LIN {X 0,Y 227.562,Z 874.921,A -85,B 0,C 180,E1 18435.228,E2 18435.228} C_VEL
LIN {X 0,Y 232.413,Z 908.174,A -85,B 0,C 180,E1 18441.181,E2 18441.181} C_VEL
LIN {X 0,Y 223.238,Z 943.271,A -85,B 0,C 180,E1 18449.512,E2 18449.512} C_VEL
LIN {X 0,Y 216.658,Z 965.158,A -85,B 0,C 180,E1 18460.084,E2 18460.084} C_VEL
LIN {X 0,Y 215.346,Z 974.266,A -85,B 0,C 180,E1 18472.803,E2 18472.803} C_VEL
LIN {X 0,Y 221.79,Z 968.351,A -85,B 0,C 180,E1 18485.562,E2 18485.562} C_VEL
LIN {X 0,Y 234.33,Z 948.382,A -85,B 0,C 180,E1 18496.092,E2 18496.092} C_VEL
LIN {X 0,Y 246.199,Z 920.964,A -85,B 0,C 180,E1 18503.2,E2 18503.2} C_VEL
LIN {X 0,Y 242.131,Z 889.578,A -85,B 0,C 180,E1 18511.964,E2 18511.964} C_VEL
LIN {X 0,Y 229.382,Z 860.327,A -85,B 0,C 180,E1 18522.556,E2 18522.556} C_VEL
LIN {X 0,Y 219.392,Z 845.564,A -85,B 0,C 180,E1 18532.052,E2 18532.052} C_VEL
LIN {X 0,Y 215.629,Z 839.103,A -85,B 0,C 180,E1 18538.996,E2 18538.996} C_VEL
LIN {X 0,Y 216.706,Z 841.817,A -85,B 0,C 180,E1 18553.322,E2 18553.322} C_VEL
LIN {X 0,Y 226.196,Z 855.249,A -85,B 0,C 180,E1 18564.093,E2 18564.093} C_VEL
LIN {X 0,Y 243.066,Z 883.319,A -85,B 0,C 180,E1 18574.736,E2 18574.736} C_VEL
LIN {X 0,Y 255.06,Z 918.124,A -85,B 0,C 180,E1 18582.6,E2 18582.6} C_VEL
LIN {X 0,Y 254.028,Z 931.092,A -85,B 0,C 180,E1 18584.355,E2 18584.355} C_VEL
LIN {X 0,Y 237.373,Z 975.39,A -85,B 0,C 180,E1 18590.854,E2 18590.854} C_VEL
LIN {X 0,Y 221.129,Z 1010.154,A -85,B 0,C 180,E1 18601.29,E2 18601.29} C_VEL
LIN {X 0,Y 213.42,Z 1031.37,A -85,B 0,C 180,E1 18614.546,E2 18614.546} C_VEL
LIN {X 0,Y 214.183,Z 1038.324,A -85,B 0,C 180,E1 18627.971,E2 18627.971} C_VEL
LIN {X 0,Y 213.62,Z 1033.071,A -85,B 0,C 180,E1 18638.747,E2 18638.747} C_VEL
LIN {X 0,Y 215.705,Z 1013.058,A -85,B 0,C 180,E1 18651.676,E2 18651.676} C_VEL
LIN {X 0,Y 225.346,Z 978.895,A -85,B 0,C 180,E1 18662.658,E2 18662.658} C_VEL
LIN {X 0,Y 237.301,Z 933.937,A -85,B 0,C 180,E1 18670.068,E2 18670.068} C_VEL
LIN {X 0,Y 239.733,Z 912.196,A -85,B 0,C 180,E1 18672.372,E2 18672.372} C_VEL
LIN {X 0,Y 223.495,Z 863.245,A -85,B 0,C 180,E1 18678.375,E2 18678.375} C_VEL
LIN {X 0,Y 208.076,Z 831.81,A -85,B 0,C 180,E1 18683.175,E2 18683.175} C_VEL
LIN {X 0,Y 208.641,Z 831.81,A -85,B 0,C 180,E1 18696.413,E2 18696.413} C_VEL
LIN {X 0,Y 209.995,Z 831.81,A -85,B 0,C 180,E1 18709.587,E2 18709.587} C_VEL
LIN {X 0,Y 211.06,Z 831.81,A -85,B 0,C 180,E1 18722.056,E2 18722.056} C_VEL
LIN {X 0,Y 209.619,Z 831.81,A -85,B 0,C 180,E1 18734.674,E2 18734.674} C_VEL
LIN {X 0,Y 208.453,Z 831.81,A -85,B 0,C 180,E1 18748.239,E2 18748.239} C_VEL
LIN {X 0,Y 207.773,Z 831.81,A -85,B 0,C 180,E1 18755.093,E2 18755.093} C_VEL
LIN {X 0,Y 199.619,Z 831.81,A -85,B 0,C 180,E1 18764.876,E2 18764.876} C_VEL
LIN {X 0,Y 200.129,Z 831.81,A -85,B 0,C 180,E1 18780.692,E2 18780.692} C_VEL
LIN {X 0,Y 200.595,Z 833.153,A -85,B 0,C 180,E1 18786.258,E2 18786.258} C_VEL
LIN {X 0,Y 220.002,Z 874.825,A -85,B 0,C 180,E1 18793.82,E2 18793.82} C_VEL
LIN {X 0,Y 225.22,Z 909.27,A -85,B 0,C 180,E1 18800.302,E2 18800.302} C_VEL
LIN {X 0,Y 215.598,Z 944.601,A -85,B 0,C 180,E1 18808.991,E2 18808.991} C_VEL
LIN {X 0,Y 208.485,Z 967.346,A -85,B 0,C 180,E1 18820.692,E2 18820.692} C_VEL
LIN {X 0,Y 207.716,Z 975.562,A -85,B 0,C 180,E1 18834.047,E2 18834.047} C_VEL
LIN {X 0,Y 214.927,Z 969.025,A -85,B 0,C 180,E1 18846.881,E2 18846.881} C_VEL
LIN {X 0,Y 228.472,Z 948.449,A -85,B 0,C 180,E1 18857.625,E2 18857.625} C_VEL
LIN {X 0,Y 239.818,Z 923.429,A -85,B 0,C 180,E1 18864.258,E2 18864.258} C_VEL
LIN {X 0,Y 236.55,Z 893.1,A -85,B 0,C 180,E1 18873.318,E2 18873.318} C_VEL
LIN {X 0,Y 225.614,Z 866.279,A -85,B 0,C 180,E1 18883.894,E2 18883.894} C_VEL
LIN {X 0,Y 217.441,Z 852.723,A -85,B 0,C 180,E1 18893.114,E2 18893.114} C_VEL
LIN {X 0,Y 214.592,Z 847.026,A -85,B 0,C 180,E1 18898.991,E2 18898.991} C_VEL
LIN {X 0,Y 215.401,Z 849.582,A -85,B 0,C 180,E1 18912.822,E2 18912.822} C_VEL
LIN {X 0,Y 224.366,Z 863.156,A -85,B 0,C 180,E1 18923.623,E2 18923.623} C_VEL
LIN {X 0,Y 239.322,Z 890.023,A -85,B 0,C 180,E1 18934.117,E2 18934.117} C_VEL
LIN {X 0,Y 249.469,Z 923.65,A -85,B 0,C 180,E1 18942.061,E2 18942.061} C_VEL
LIN {X 0,Y 234.402,Z 967.505,A -85,B 0,C 180,E1 18948.127,E2 18948.127} C_VEL
LIN {X 0,Y 217.225,Z 1002.987,A -85,B 0,C 180,E1 18957.642,E2 18957.642} C_VEL
LIN {X 0,Y 206.636,Z 1026.774,A -85,B 0,C 180,E1 18970.703,E2 18970.703} C_VEL
LIN {X 0,Y 205.698,Z 1036.793,A -85,B 0,C 180,E1 18984.937,E2 18984.937} C_VEL
LIN {X 0,Y 205.898,Z 1033.928,A -85,B 0,C 180,E1 18996.348,E2 18996.348} C_VEL
LIN {X 0,Y 206.967,Z 1016.698,A -85,B 0,C 180,E1 19009.824,E2 19009.824} C_VEL
LIN {X 0,Y 215.978,Z 984.595,A -85,B 0,C 180,E1 19021.802,E2 19021.802} C_VEL
LIN {X 0,Y 228.47,Z 941.098,A -85,B 0,C 180,E1 19030.075,E2 19030.075} C_VEL
LIN {X 0,Y 232.456,Z 913.301,A -85,B 0,C 180,E1 19033.274,E2 19033.274} C_VEL
LIN {X 0,Y 216.734,Z 865.176,A -85,B 0,C 180,E1 19039.626,E2 19039.626} C_VEL
LIN {X 0,Y 200.024,Z 831.81,A -85,B 0,C 180,E1 19045.311,E2 19045.311} C_VEL
LIN {X 0,Y 201.036,Z 831.81,A -85,B 0,C 180,E1 19060.663,E2 19060.663} C_VEL
LIN {X 0,Y 202.402,Z 831.81,A -85,B 0,C 180,E1 19073.538,E2 19073.538} C_VEL
LIN {X 0,Y 202.406,Z 831.81,A -85,B 0,C 180,E1 19086.453,E2 19086.453} C_VEL
LIN {X 0,Y 201.019,Z 831.81,A -85,B 0,C 180,E1 19099.856,E2 19099.856} C_VEL
LIN {X 0,Y 199.779,Z 831.81,A -85,B 0,C 180,E1 19115.035,E2 19115.035} C_VEL
LIN {X 0,Y 199.619,Z 831.81,A -85,B 0,C 180,E1 19124.876,E2 19124.876} C_VEL
LIN {X 0,Y 191.641,Z 831.81,A -85,B 0,C 180,E1 19135.041,E2 19135.041} C_VEL
LIN {X 0,Y 192.321,Z 833.227,A -85,B 0,C 180,E1 19144.01,E2 19144.01} C_VEL
LIN {X 0,Y 212.038,Z 873.85,A -85,B 0,C 180,E1 19152.114,E2 19152.114} C_VEL
LIN {X 0,Y 218.056,Z 907.218,A -85,B 0,C 180,E1 19158.702,E2 19158.702} C_VEL
LIN {X 0,Y 210.506,Z 938.161,A -85,B 0,C 180,E1 19165.865,E2 19165.865} C_VEL
LIN {X 0,Y 202.25,Z 962.969,A -85,B 0,C 180,E1 19176.462,E2 19176.462} C_VEL
LIN {X 0,Y 199.165,Z 975.841,A -85,B 0,C 180,E1 19190.051,E2 19190.051} C_VEL
LIN {X 0,Y 204.368,Z 973.813,A -85,B 0,C 180,E1 19203.842,E2 19203.842} C_VEL
LIN {X 0,Y 217.789,Z 956.53,A -85,B 0,C 180,E1 19216.152,E2 19216.152} C_VEL
LIN {X 0,Y 233.487,Z 926.207,A -85,B 0,C 180,E1 19225.271,E2 19225.271} C_VEL
LIN {X 0,Y 231.391,Z 897.943,A -85,B 0,C 180,E1 19234.249,E2 19234.249} C_VEL
LIN {X 0,Y 222.035,Z 872.175,A -85,B 0,C 180,E1 19245.152,E2 19245.152} C_VEL
LIN {X 0,Y 215.105,Z 859.024,A -85,B 0,C 180,E1 19254.818,E2 19254.818} C_VEL
LIN {X 0,Y 213.156,Z 854.83,A -85,B 0,C 180,E1 19260.004,E2 19260.004} C_VEL
LIN {X 0,Y 214.206,Z 857.664,A -85,B 0,C 180,E1 19272.602,E2 19272.602} C_VEL
LIN {X 0,Y 222.658,Z 871.543,A -85,B 0,C 180,E1 19283.498,E2 19283.498} C_VEL
LIN {X 0,Y 235.877,Z 897.817,A -85,B 0,C 180,E1 19293.883,E2 19293.883} C_VEL
LIN {X 0,Y 243.66,Z 928.776,A -85,B 0,C 180,E1 19301.455,E2 19301.455} C_VEL
LIN {X 0,Y 225.466,Z 973.136,A -85,B 0,C 180,E1 19308.014,E2 19308.014} C_VEL
LIN {X 0,Y 207.536,Z 1007.322,A -85,B 0,C 180,E1 19318.602,E2 19318.602} C_VEL
LIN {X 0,Y 198.142,Z 1027.993,A -85,B 0,C 180,E1 19332.014,E2 19332.014} C_VEL
LIN {X 0,Y 197.604,Z 1035.315,A -85,B 0,C 180,E1 19343.386,E2 19343.386} C_VEL
LIN {X 0,Y 198.026,Z 1033.573,A -85,B 0,C 180,E1 19354.984,E2 19354.984} C_VEL
LIN {X 0,Y 198.809,Z 1017.493,A -85,B 0,C 180,E1 19369.18,E2 19369.18} C_VEL
LIN {X 0,Y 207.283,Z 987.806,A -85,B 0,C 180,E1 19381.442,E2 19381.442} C_VEL
LIN {X 0,Y 219.997,Z 945.926,A -85,B 0,C 180,E1 19390.293,E2 19390.293} C_VEL
LIN {X 0,Y 225.514,Z 915.954,A -85,B 0,C 180,E1 19394.003,E2 19394.003} C_VEL
LIN {X 0,Y 210.731,Z 868.772,A -85,B 0,C 180,E1 19400.705,E2 19400.705} C_VEL
LIN {X 0,Y 191.908,Z 831.81,A -85,B 0,C 180,E1 19407.681,E2 19407.681} C_VEL
LIN {X 0,Y 193.242,Z 831.81,A -85,B 0,C 180,E1 19424.041,E2 19424.041} C_VEL
LIN {X 0,Y 194.824,Z 831.81,A -85,B 0,C 180,E1 19437.763,E2 19437.763} C_VEL
LIN {X 0,Y 193.764,Z 831.81,A -85,B 0,C 180,E1 19451.763,E2 19451.763} C_VEL
LIN {X 0,Y 192.436,Z 831.81,A -85,B 0,C 180,E1 19465.701,E2 19465.701} C_VEL
LIN {X 0,Y 191.599,Z 831.81,A -85,B 0,C 180,E1 19482.314,E2 19482.314} C_VEL
LIN {X 0,Y 191.641,Z 831.81,A -85,B 0,C 180,E1 19495.041,E2 19495.041} C_VEL
LIN {X 0,Y 183.76,Z 831.81,A -85,B 0,C 180,E1 19499.036,E2 19499.036} C_VEL
LIN {X 0,Y 184.366,Z 834.043,A -85,B 0,C 180,E1 19501.623,E2 19501.623} C_VEL
LIN {X 0,Y 204.05,Z 872.307,A -85,B 0,C 180,E1 19510.187,E2 19510.187} C_VEL
LIN {X 0,Y 211.019,Z 906.88,A -85,B 0,C 180,E1 19517.363,E2 19517.363} C_VEL
LIN {X 0,Y 204.912,Z 934.231,A -85,B 0,C 180,E1 19523.621,E2 19523.621} C_VEL
LIN {X 0,Y 195.354,Z 961.456,A -85,B 0,C 180,E1 19534.455,E2 19534.455} C_VEL
LIN {X 0,Y 191.182,Z 976.246,A -85,B 0,C 180,E1 19548.467,E2 19548.467} C_VEL
LIN {X 0,Y 195.705,Z 976.136,A -85,B 0,C 180,E1 19562.873,E2 19562.873} C_VEL
LIN {X 0,Y 208.443,Z 961.663,A -85,B 0,C 180,E1 19575.466,E2 19575.466} C_VEL
LIN {X 0,Y 225.666,Z 934.091,A -85,B 0,C 180,E1 19584.848,E2 19584.848} C_VEL
LIN {X 0,Y 227.198,Z 909.123,A -85,B 0,C 180,E1 19592.935,E2 19592.935} C_VEL
LIN {X 0,Y 220.603,Z 883.227,A -85,B 0,C 180,E1 19603.518,E2 19603.518} C_VEL
LIN {X 0,Y 213.521,Z 867.423,A -85,B 0,C 180,E1 19614.523,E2 19614.523} C_VEL
LIN {X 0,Y 211.564,Z 862.576,A -85,B 0,C 180,E1 19621.051,E2 19621.051} C_VEL
LIN {X 0,Y 212.721,Z 865.53,A -85,B 0,C 180,E1 19632.238,E2 19632.238} C_VEL
LIN {X 0,Y 220.513,Z 879.568,A -85,B 0,C 180,E1 19643.316,E2 19643.316} C_VEL
LIN {X 0,Y 232.182,Z 905.731,A -85,B 0,C 180,E1 19653.756,E2 19653.756} C_VEL
LIN {X 0,Y 236.869,Z 933.02,A -85,B 0,C 180,E1 19660.477,E2 19660.477} C_VEL
LIN {X 0,Y 217.79,Z 975.94,A -85,B 0,C 180,E1 19667.34,E2 19667.34} C_VEL
LIN {X 0,Y 199.319,Z 1008.691,A -85,B 0,C 180,E1 19678.438,E2 19678.438} C_VEL
LIN {X 0,Y 189.668,Z 1029.12,A -85,B 0,C 180,E1 19693.739,E2 19693.739} C_VEL
LIN {X 0,Y 190.322,Z 1034.634,A -85,B 0,C 180,E1 19707.716,E2 19707.716} C_VEL
LIN {X 0,Y 189.648,Z 1028.232,A -85,B 0,C 180,E1 19720.373,E2 19720.373} C_VEL
LIN {X 0,Y 192.94,Z 1007.535,A -85,B 0,C 180,E1 19734.39,E2 19734.39} C_VEL
LIN {X 0,Y 204.321,Z 973.033,A -85,B 0,C 180,E1 19746.036,E2 19746.036} C_VEL
LIN {X 0,Y 217.585,Z 928.052,A -85,B 0,C 180,E1 19753.569,E2 19753.569} C_VEL
LIN {X 0,Y 216.675,Z 909.509,A -85,B 0,C 180,E1 19756.189,E2 19756.189} C_VEL
LIN {X 0,Y 200.96,Z 864.247,A -85,B 0,C 180,E1 19763.171,E2 19763.171} C_VEL
LIN {X 0,Y 183.937,Z 831.81,A -85,B 0,C 180,E1 19770.031,E2 19770.031} C_VEL
LIN {X 0,Y 185.067,Z 831.81,A -85,B 0,C 180,E1 19783.316,E2 19783.316} C_VEL
LIN {X 0,Y 186.796,Z 831.81,A -85,B 0,C 180,E1 19797.667,E2 19797.667} C_VEL
LIN {X 0,Y 185.759,Z 831.81,A -85,B 0,C 180,E1 19811.781,E2 19811.781} C_VEL
LIN {X 0,Y 184.165,Z 831.81,A -85,B 0,C 180,E1 19826.946,E2 19826.946} C_VEL
LIN {X 0,Y 183.391,Z 831.81,A -85,B 0,C 180,E1 19844.695,E2 19844.695} C_VEL
LIN {X 0,Y 183.76,Z 831.81,A -85,B 0,C 180,E1 19859.036,E2 19859.036} C_VEL
LIN {X 0,Y 186.391,Z 840.3,A -85,B 0,C 180,E1 19862.564,E2 19862.564} C_VEL
LIN {X 0,Y 191.215,Z 859.617,A -85,B 0,C 180,E1 19865.511,E2 19865.511} C_VEL
LIN {X 0,Y 202.871,Z 896.426,A -85,B 0,C 180,E1 19873.655,E2 19873.655} C_VEL
LIN {X 0,Y 201.758,Z 923.575,A -85,B 0,C 180,E1 19879.766,E2 19879.766} C_VEL
LIN {X 0,Y 190.423,Z 955.55,A -85,B 0,C 180,E1 19890.234,E2 19890.234} C_VEL
LIN {X 0,Y 183.892,Z 973.75,A -85,B 0,C 180,E1 19903.116,E2 19903.116} C_VEL
LIN {X 0,Y 184.79,Z 979.219,A -85,B 0,C 180,E1 19916.85,E2 19916.85} C_VEL
LIN {X 0,Y 195.139,Z 970.902,A -85,B 0,C 180,E1 19931.377,E2 19931.377} C_VEL
LIN {X 0,Y 212.061,Z 948.596,A -85,B 0,C 180,E1 19942.634,E2 19942.634} C_VEL
LIN {X 0,Y 221.068,Z 930.986,A -85,B 0,C 180,E1 19947.718,E2 19947.718} C_VEL
LIN {X 0,Y 220.618,Z 904.893,A -85,B 0,C 180,E1 19957.239,E2 19957.239} C_VEL
LIN {X 0,Y 214.239,Z 881.983,A -85,B 0,C 180,E1 19968.771,E2 19968.771} C_VEL
LIN {X 0,Y 210.112,Z 870.509,A -85,B 0,C 180,E1 19980.042,E2 19980.042} C_VEL
LIN {X 0,Y 210.899,Z 873.271,A -85,B 0,C 180,E1 19991.888,E2 19991.888} C_VEL
LIN {X 0,Y 218.414,Z 888.041,A -85,B 0,C 180,E1 20003.553,E2 20003.553} C_VEL
LIN {X 0,Y 228.665,Z 915.907,A -85,B 0,C 180,E1 20014.347,E2 20014.347} C_VEL
LIN {X 0,Y 230.466,Z 936.14,A -85,B 0,C 180,E1 20019.335,E2 20019.335} C_VEL
LIN {X 0,Y 210.034,Z 978.625,A -85,B 0,C 180,E1 20026.656,E2 20026.656} C_VEL
LIN {X 0,Y 190.468,Z 1010.936,A -85,B 0,C 180,E1 20038.811,E2 20038.811} C_VEL
LIN {X 0,Y 181.65,Z 1028.735,A -85,B 0,C 180,E1 20053.919,E2 20053.919} C_VEL
LIN {X 0,Y 182.379,Z 1033.404,A -85,B 0,C 180,E1 20067.616,E2 20067.616} C_VEL
LIN {X 0,Y 181.7,Z 1026.762,A -85,B 0,C 180,E1 20080.832,E2 20080.832} C_VEL
LIN {X 0,Y 185.957,Z 1004.434,A -85,B 0,C 180,E1 20096.014,E2 20096.014} C_VEL
LIN {X 0,Y 198.195,Z 968.996,A -85,B 0,C 180,E1 20107.775,E2 20107.775} C_VEL
LIN {X 0,Y 211.623,Z 924.475,A -85,B 0,C 180,E1 20115.054,E2 20115.054} C_VEL
LIN {X 0,Y 200.47,Z 879.884,A -85,B 0,C 180,E1 20122.338,E2 20122.338} C_VEL
LIN {X 0,Y 177.724,Z 836.816,A -85,B 0,C 180,E1 20131.478,E2 20131.478} C_VEL
LIN {X 0,Y 176.108,Z 831.81,A -85,B 0,C 180,E1 20133.375,E2 20133.375} C_VEL
LIN {X 0,Y 177.694,Z 831.81,A -85,B 0,C 180,E1 20149.153,E2 20149.153} C_VEL
LIN {X 0,Y 178.887,Z 831.81,A -85,B 0,C 180,E1 20162.426,E2 20162.426} C_VEL
LIN {X 0,Y 177.05,Z 831.81,A -85,B 0,C 180,E1 20177.453,E2 20177.453} C_VEL
LIN {X 0,Y 175.466,Z 831.81,A -85,B 0,C 180,E1 20194.752,E2 20194.752} C_VEL
LIN {X 0,Y 175.214,Z 831.81,A -85,B 0,C 180,E1 20209.489,E2 20209.489} C_VEL
LIN {X 0,Y 175.909,Z 833.4,A -85,B 0,C 180,E1 20218.619,E2 20218.619} C_VEL
LIN {X 0,Y 191.215,Z 859.617,A -85,B 0,C 180,E1 20225.511,E2 20225.511} C_VEL
LIN {X 0,Y 194.584,Z 890.587,A -85,B 0,C 180,E1 20230.688,E2 20230.688} C_VEL
LIN {X 0,Y 196.142,Z 919.972,A -85,B 0,C 180,E1 20237.682,E2 20237.682} C_VEL
LIN {X 0,Y 184.288,Z 952.559,A -85,B 0,C 180,E1 20247.639,E2 20247.639} C_VEL
LIN {X 0,Y 176.603,Z 972.923,A -85,B 0,C 180,E1 20260.827,E2 20260.827} C_VEL
LIN {X 0,Y 176.358,Z 980.408,A -85,B 0,C 180,E1 20275.381,E2 20275.381} C_VEL
LIN {X 0,Y 186.157,Z 974.124,A -85,B 0,C 180,E1 20290.7,E2 20290.7} C_VEL
LIN {X 0,Y 203.973,Z 952.978,A -85,B 0,C 180,E1 20303.022,E2 20303.022} C_VEL
LIN {X 0,Y 214.807,Z 934.604,A -85,B 0,C 180,E1 20308.603,E2 20308.603} C_VEL
LIN {X 0,Y 215.408,Z 908.684,A -85,B 0,C 180,E1 20318.754,E2 20318.754} C_VEL
LIN {X 0,Y 210.36,Z 886.921,A -85,B 0,C 180,E1 20330.924,E2 20330.924} C_VEL
LIN {X 0,Y 207.86,Z 878.109,A -85,B 0,C 180,E1 20341.069,E2 20341.069} C_VEL
LIN {X 0,Y 208.777,Z 881.102,A -85,B 0,C 180,E1 20351.72,E2 20351.72} C_VEL
LIN {X 0,Y 215.062,Z 894.834,A -85,B 0,C 180,E1 20362.842,E2 20362.842} C_VEL
LIN {X 0,Y 223.556,Z 921.192,A -85,B 0,C 180,E1 20373.557,E2 20373.557} C_VEL
LIN {X 0,Y 224.375,Z 938.538,A -85,B 0,C 180,E1 20378.048,E2 20378.048} C_VEL
LIN {X 0,Y 203.144,Z 979.828,A -85,B 0,C 180,E1 20385.547,E2 20385.547} C_VEL
LIN {X 0,Y 183.512,Z 1010.068,A -85,B 0,C 180,E1 20397.486,E2 20397.486} C_VEL
LIN {X 0,Y 173.735,Z 1027.925,A -85,B 0,C 180,E1 20413.629,E2 20413.629} C_VEL
LIN {X 0,Y 174.42,Z 1032.164,A -85,B 0,C 180,E1 20427.508,E2 20427.508} C_VEL
LIN {X 0,Y 173.775,Z 1025.269,A -85,B 0,C 180,E1 20441.333,E2 20441.333} C_VEL
LIN {X 0,Y 178.466,Z 1002.921,A -85,B 0,C 180,E1 20456.959,E2 20456.959} C_VEL
LIN {X 0,Y 191.33,Z 967.485,A -85,B 0,C 180,E1 20469.019,E2 20469.019} C_VEL
LIN {X 0,Y 204.435,Z 922.73,A -85,B 0,C 180,E1 20476.56,E2 20476.56} C_VEL
LIN {X 0,Y 192.469,Z 878.492,A -85,B 0,C 180,E1 20484.437,E2 20484.437} C_VEL
LIN {X 0,Y 170.224,Z 837.238,A -85,B 0,C 180,E1 20494.343,E2 20494.343} C_VEL
LIN {X 0,Y 168.192,Z 831.81,A -85,B 0,C 180,E1 20496.038,E2 20496.038} C_VEL
LIN {X 0,Y 170.066,Z 831.81,A -85,B 0,C 180,E1 20512.302,E2 20512.302} C_VEL
LIN {X 0,Y 170.826,Z 831.81,A -85,B 0,C 180,E1 20522.541,E2 20522.541} C_VEL
LIN {X 0,Y 168.685,Z 831.81,A -85,B 0,C 180,E1 20539.156,E2 20539.156} C_VEL
LIN {X 0,Y 167.239,Z 831.81,A -85,B 0,C 180,E1 20556.14,E2 20556.14} C_VEL
LIN {X 0,Y 167.192,Z 831.81,A -85,B 0,C 180,E1 20573.843,E2 20573.843} C_VEL
LIN {X 0,Y 171.42,Z 838.812,A -85,B 0,C 180,E1 20577.243,E2 20577.243} C_VEL
LIN {X 0,Y 190.329,Z 875.774,A -85,B 0,C 180,E1 20587.202,E2 20587.202} C_VEL
LIN {X 0,Y 194.584,Z 890.587,A -85,B 0,C 180,E1 20590.688,E2 20590.688} C_VEL
LIN {X 0,Y 189.38,Z 920.442,A -85,B 0,C 180,E1 20596.395,E2 20596.395} C_VEL
LIN {X 0,Y 176.73,Z 953.815,A -85,B 0,C 180,E1 20606.923,E2 20606.923} C_VEL
LIN {X 0,Y 168.432,Z 974.957,A -85,B 0,C 180,E1 20621.572,E2 20621.572} C_VEL
LIN {X 0,Y 168.055,Z 981.354,A -85,B 0,C 180,E1 20633.975,E2 20633.975} C_VEL
LIN {X 0,Y 177.219,Z 977.055,A -85,B 0,C 180,E1 20649.957,E2 20649.957} C_VEL
LIN {X 0,Y 195.61,Z 957.528,A -85,B 0,C 180,E1 20663.252,E2 20663.252} C_VEL
LIN {X 0,Y 208.733,Z 937.243,A -85,B 0,C 180,E1 20669.877,E2 20669.877} C_VEL
LIN {X 0,Y 210.279,Z 913.272,A -85,B 0,C 180,E1 20679.956,E2 20679.956} C_VEL
LIN {X 0,Y 206.874,Z 892.397,A -85,B 0,C 180,E1 20692.523,E2 20692.523} C_VEL
LIN {X 0,Y 205.263,Z 885.655,A -85,B 0,C 180,E1 20703.57,E2 20703.57} C_VEL
LIN {X 0,Y 206.622,Z 889.914,A -85,B 0,C 180,E1 20712.734,E2 20712.734} C_VEL
LIN {X 0,Y 213.581,Z 907.162,A -85,B 0,C 180,E1 20725.187,E2 20725.187} C_VEL
LIN {X 0,Y 219.301,Z 935.054,A -85,B 0,C 180,E1 20735.426,E2 20735.426} C_VEL
LIN {X 0,Y 214.716,Z 948.635,A -85,B 0,C 180,E1 20737.751,E2 20737.751} C_VEL
LIN {X 0,Y 192.177,Z 987.241,A -85,B 0,C 180,E1 20746.296,E2 20746.296} C_VEL
LIN {X 0,Y 172.857,Z 1014.546,A -85,B 0,C 180,E1 20759.683,E2 20759.683} C_VEL
LIN {X 0,Y 165.41,Z 1028.821,A -85,B 0,C 180,E1 20776.742,E2 20776.742} C_VEL
LIN {X 0,Y 166.469,Z 1030.898,A -85,B 0,C 180,E1 20787.388,E2 20787.388} C_VEL
LIN {X 0,Y 165.859,Z 1024.867,A -85,B 0,C 180,E1 20800.545,E2 20800.545} C_VEL
LIN {X 0,Y 170.564,Z 1002.702,A -85,B 0,C 180,E1 20817.347,E2 20817.347} C_VEL
LIN {X 0,Y 184.138,Z 967.014,A -85,B 0,C 180,E1 20830.081,E2 20830.081} C_VEL
LIN {X 0,Y 197.174,Z 923.474,A -85,B 0,C 180,E1 20837.775,E2 20837.775} C_VEL
LIN {X 0,Y 185.721,Z 879.825,A -85,B 0,C 180,E1 20846.167,E2 20846.167} C_VEL
LIN {X 0,Y 163.7,Z 838.437,A -85,B 0,C 180,E1 20857.151,E2 20857.151} C_VEL
LIN {X 0,Y 160.411,Z 831.81,A -85,B 0,C 180,E1 20859.901,E2 20859.901} C_VEL
LIN {X 0,Y 162.637,Z 831.81,A -85,B 0,C 180,E1 20877.32,E2 20877.32} C_VEL
LIN {X 0,Y 161.668,Z 831.81,A -85,B 0,C 180,E1 20889.726,E2 20889.726} C_VEL
LIN {X 0,Y 159.923,Z 831.81,A -85,B 0,C 180,E1 20905.646,E2 20905.646} C_VEL
LIN {X 0,Y 159.089,Z 831.81,A -85,B 0,C 180,E1 20924.321,E2 20924.321} C_VEL
LIN {X 0,Y 159.263,Z 833.311,A -85,B 0,C 180,E1 20931.205,E2 20931.205} C_VEL
LIN {X 0,Y 179.534,Z 867.301,A -85,B 0,C 180,E1 20942.84,E2 20942.84} C_VEL
LIN {X 0,Y 189.462,Z 902.527,A -85,B 0,C 180,E1 20951.836,E2 20951.836} C_VEL
LIN {X 0,Y 189.38,Z 920.442,A -85,B 0,C 180,E1 20956.395,E2 20956.395} C_VEL
LIN {X 0,Y 172.851,Z 945.942,A -85,B 0,C 180,E1 20962.211,E2 20962.211} C_VEL
LIN {X 0,Y 162.778,Z 969.908,A -85,B 0,C 180,E1 20975.348,E2 20975.348} C_VEL
LIN {X 0,Y 159.539,Z 981.079,A -85,B 0,C 180,E1 20989.445,E2 20989.445} C_VEL
LIN {X 0,Y 166.016,Z 981.123,A -85,B 0,C 180,E1 21006.451,E2 21006.451} C_VEL
LIN {X 0,Y 181.974,Z 967.476,A -85,B 0,C 180,E1 21020.477,E2 21020.477} C_VEL
LIN {X 0,Y 202.508,Z 940.831,A -85,B 0,C 180,E1 21030.853,E2 21030.853} C_VEL
LIN {X 0,Y 205.212,Z 918.002,A -85,B 0,C 180,E1 21041.127,E2 21041.127} C_VEL
LIN {X 0,Y 203.308,Z 898.889,A -85,B 0,C 180,E1 21053.575,E2 21053.575} C_VEL
LIN {X 0,Y 202.664,Z 893.141,A -85,B 0,C 180,E1 21062.15,E2 21062.15} C_VEL
LIN {X 0,Y 203.409,Z 895.743,A -85,B 0,C 180,E1 21070.754,E2 21070.754} C_VEL
LIN {X 0,Y 209.217,Z 912.813,A -85,B 0,C 180,E1 21084.142,E2 21084.142} C_VEL
LIN {X 0,Y 213.52,Z 939.074,A -85,B 0,C 180,E1 21094.416,E2 21094.416} C_VEL
LIN {X 0,Y 191.165,Z 979.737,A -85,B 0,C 180,E1 21102.445,E2 21102.445} C_VEL
LIN {X 0,Y 168.467,Z 1010.205,A -85,B 0,C 180,E1 21115.738,E2 21115.738} C_VEL
LIN {X 0,Y 157.846,Z 1026.472,A -85,B 0,C 180,E1 21133.336,E2 21133.336} C_VEL
LIN {X 0,Y 158.506,Z 1029.621,A -85,B 0,C 180,E1 21147.257,E2 21147.257} C_VEL
LIN {X 0,Y 157.901,Z 1023.383,A -85,B 0,C 180,E1 21161.083,E2 21161.083} C_VEL
LIN {X 0,Y 162.845,Z 1001.902,A -85,B 0,C 180,E1 21178.048,E2 21178.048} C_VEL
LIN {X 0,Y 177.022,Z 966.525,A -85,B 0,C 180,E1 21191.226,E2 21191.226} C_VEL
LIN {X 0,Y 190.142,Z 924.965,A -85,B 0,C 180,E1 21198.919,E2 21198.919} C_VEL
LIN {X 0,Y 179.743,Z 883.078,A -85,B 0,C 180,E1 21207.608,E2 21207.608} C_VEL
LIN {X 0,Y 159.842,Z 844.651,A -85,B 0,C 180,E1 21218.59,E2 21218.59} C_VEL
LIN {X 0,Y 152.802,Z 831.81,A -85,B 0,C 180,E1 21224.54,E2 21224.54} C_VEL
LIN {X 0,Y 154.572,Z 831.81,A -85,B 0,C 180,E1 21237.181,E2 21237.181} C_VEL
LIN {X 0,Y 153.876,Z 831.81,A -85,B 0,C 180,E1 21248.502,E2 21248.502} C_VEL
LIN {X 0,Y 151.697,Z 831.81,A -85,B 0,C 180,E1 21266.75,E2 21266.75} C_VEL
LIN {X 0,Y 151.22,Z 833.485,A -85,B 0,C 180,E1 21286.446,E2 21286.446} C_VEL
LIN {X 0,Y 171.682,Z 866.232,A -85,B 0,C 180,E1 21299.917,E2 21299.917} C_VEL
LIN {X 0,Y 182.215,Z 900.964,A -85,B 0,C 180,E1 21309.635,E2 21309.635} C_VEL
LIN {X 0,Y 181.293,Z 925.36,A -85,B 0,C 180,E1 21316.074,E2 21316.074} C_VEL
LIN {X 0,Y 172.851,Z 945.942,A -85,B 0,C 180,E1 21322.211,E2 21322.211} C_VEL
LIN {X 0,Y 157.204,Z 965.88,A -85,B 0,C 180,E1 21330.895,E2 21330.895} C_VEL
LIN {X 0,Y 151.596,Z 981.519,A -85,B 0,C 180,E1 21348.02,E2 21348.02} C_VEL
LIN {X 0,Y 156.618,Z 983.373,A -85,B 0,C 180,E1 21364.558,E2 21364.558} C_VEL
LIN {X 0,Y 172.816,Z 971.635,A -85,B 0,C 180,E1 21380.143,E2 21380.143} C_VEL
LIN {X 0,Y 194.93,Z 946.608,A -85,B 0,C 180,E1 21391.138,E2 21391.138} C_VEL
LIN {X 0,Y 199.874,Z 927.047,A -85,B 0,C 180,E1 21400.025,E2 21400.025} C_VEL
LIN {X 0,Y 199.733,Z 907.787,A -85,B 0,C 180,E1 21412.363,E2 21412.363} C_VEL
LIN {X 0,Y 199.604,Z 900.564,A -85,B 0,C 180,E1 21422.183,E2 21422.183} C_VEL
LIN {X 0,Y 200.327,Z 903.418,A -85,B 0,C 180,E1 21430.922,E2 21430.922} C_VEL
LIN {X 0,Y 204.851,Z 918.959,A -85,B 0,C 180,E1 21443.416,E2 21443.416} C_VEL
LIN {X 0,Y 207.695,Z 942.544,A -85,B 0,C 180,E1 21453.237,E2 21453.237} C_VEL
LIN {X 0,Y 183.218,Z 982.719,A -85,B 0,C 180,E1 21461.64,E2 21461.64} C_VEL
LIN {X 0,Y 160.271,Z 1011.071,A -85,B 0,C 180,E1 21475.382,E2 21475.382} C_VEL
LIN {X 0,Y 149.608,Z 1026.553,A -85,B 0,C 180,E1 21495.311,E2 21495.311} C_VEL
LIN {X 0,Y 150.54,Z 1028.339,A -85,B 0,C 180,E1 21507.112,E2 21507.112} C_VEL
LIN {X 0,Y 149.958,Z 1021.876,A -85,B 0,C 180,E1 21521.678,E2 21521.678} C_VEL
LIN {X 0,Y 155.739,Z 999.656,A -85,B 0,C 180,E1 21539.598,E2 21539.598} C_VEL
LIN {X 0,Y 170.937,Z 963.822,A -85,B 0,C 180,E1 21553.039,E2 21553.039} C_VEL
LIN {X 0,Y 183.119,Z 925.785,A -85,B 0,C 180,E1 21560.294,E2 21560.294} C_VEL
LIN {X 0,Y 173.229,Z 884.577,A -85,B 0,C 180,E1 21569.564,E2 21569.564} C_VEL
LIN {X 0,Y 155.112,Z 849.203,A -85,B 0,C 180,E1 21580.768,E2 21580.768} C_VEL
LIN {X 0,Y 145.374,Z 831.81,A -85,B 0,C 180,E1 21589.466,E2 21589.466} C_VEL
LIN {X 0,Y 146.631,Z 831.81,A -85,B 0,C 180,E1 21602.96,E2 21602.96} C_VEL
LIN {X 0,Y 144.079,Z 831.81,A -85,B 0,C 180,E1 21621.627,E2 21621.627} C_VEL
LIN {X 0,Y 143.084,Z 833.732,A -85,B 0,C 180,E1 21640.113,E2 21640.113} C_VEL
LIN {X 0,Y 160.324,Z 858.922,A -85,B 0,C 180,E1 21654.146,E2 21654.146} C_VEL
LIN {X 0,Y 173.3,Z 891.07,A -85,B 0,C 180,E1 21664.801,E2 21664.801} C_VEL
LIN {X 0,Y 175.854,Z 921.668,A -85,B 0,C 180,E1 21673.558,E2 21673.558} C_VEL
LIN {X 0,Y 162.234,Z 954.979,A -85,B 0,C 180,E1 21684.632,E2 21684.632} C_VEL
LIN {X 0,Y 157.204,Z 965.88,A -85,B 0,C 180,E1 21690.895,E2 21690.895} C_VEL
LIN {X 0,Y 144.318,Z 979.388,A -85,B 0,C 180,E1 21702.421,E2 21702.421} C_VEL
LIN {X 0,Y 145.403,Z 985.27,A -85,B 0,C 180,E1 21718.011,E2 21718.011} C_VEL
LIN {X 0,Y 158.561,Z 979.311,A -85,B 0,C 180,E1 21735.872,E2 21735.872} C_VEL
LIN {X 0,Y 180.544,Z 959.166,A -85,B 0,C 180,E1 21749.236,E2 21749.236} C_VEL
LIN {X 0,Y 191.489,Z 944.109,A -85,B 0,C 180,E1 21754.758,E2 21754.758} C_VEL
LIN {X 0,Y 195.316,Z 923.131,A -85,B 0,C 180,E1 21766.214,E2 21766.214} C_VEL
LIN {X 0,Y 195.821,Z 910.136,A -85,B 0,C 180,E1 21777.827,E2 21777.827} C_VEL
LIN {X 0,Y 196.839,Z 908.843,A -85,B 0,C 180,E1 21788.656,E2 21788.656} C_VEL
LIN {X 0,Y 200.283,Z 924.966,A -85,B 0,C 180,E1 21802.689,E2 21802.689} C_VEL
LIN {X 0,Y 201.558,Z 946.648,A -85,B 0,C 180,E1 21812.12,E2 21812.12} C_VEL
LIN {X 0,Y 175.046,Z 985.726,A -85,B 0,C 180,E1 21820.862,E2 21820.862} C_VEL
LIN {X 0,Y 152.125,Z 1011.869,A -85,B 0,C 180,E1 21835,E2 21835} C_VEL
LIN {X 0,Y 141.755,Z 1025.421,A -85,B 0,C 180,E1 21854.478,E2 21854.478} C_VEL
LIN {X 0,Y 142.554,Z 1027.053,A -85,B 0,C 180,E1 21866.95,E2 21866.95} C_VEL
LIN {X 0,Y 142.054,Z 1021.443,A -85,B 0,C 180,E1 21880.776,E2 21880.776} C_VEL
LIN {X 0,Y 147.807,Z 999.604,A -85,B 0,C 180,E1 21900.06,E2 21900.06} C_VEL
LIN {X 0,Y 163.521,Z 964.43,A -85,B 0,C 180,E1 21914.111,E2 21914.111} C_VEL
LIN {X 0,Y 176.204,Z 927.515,A -85,B 0,C 180,E1 21921.547,E2 21921.547} C_VEL
LIN {X 0,Y 166.98,Z 886.378,A -85,B 0,C 180,E1 21931.564,E2 21931.564} C_VEL
LIN {X 0,Y 149.802,Z 851.746,A -85,B 0,C 180,E1 21943.757,E2 21943.757} C_VEL
LIN {X 0,Y 138.418,Z 831.81,A -85,B 0,C 180,E1 21956.851,E2 21956.851} C_VEL
LIN {X 0,Y 137.559,Z 831.81,A -85,B 0,C 180,E1 21969.519,E2 21969.519} C_VEL
LIN {X 0,Y 135.11,Z 831.846,A -85,B 0,C 180,E1 21990.203,E2 21990.203} C_VEL
LIN {X 0,Y 150.161,Z 854.866,A -85,B 0,C 180,E1 22007.973,E2 22007.973} C_VEL
LIN {X 0,Y 163.909,Z 882.78,A -85,B 0,C 180,E1 22019.678,E2 22019.678} C_VEL
LIN {X 0,Y 169.651,Z 915.413,A -85,B 0,C 180,E1 22029.918,E2 22029.918} C_VEL
LIN {X 0,Y 164.17,Z 935.534,A -85,B 0,C 180,E1 22035.583,E2 22035.583} C_VEL
LIN {X 0,Y 150.134,Z 965.738,A -85,B 0,C 180,E1 22049.275,E2 22049.275} C_VEL
LIN {X 0,Y 144.318,Z 979.388,A -85,B 0,C 180,E1 22062.421,E2 22062.421} C_VEL
LIN {X 0,Y 136.844,Z 985.991,A -85,B 0,C 180,E1 22076.311,E2 22076.311} C_VEL
LIN {X 0,Y 149.147,Z 982.353,A -85,B 0,C 180,E1 22095.06,E2 22095.06} C_VEL
LIN {X 0,Y 171.178,Z 964.708,A -85,B 0,C 180,E1 22109.302,E2 22109.302} C_VEL
LIN {X 0,Y 185.225,Z 948.298,A -85,B 0,C 180,E1 22115.607,E2 22115.607} C_VEL
LIN {X 0,Y 190.371,Z 928.544,A -85,B 0,C 180,E1 22127.182,E2 22127.182} C_VEL
LIN {X 0,Y 192.126,Z 915.951,A -85,B 0,C 180,E1 22140.005,E2 22140.005} C_VEL
LIN {X 0,Y 193.062,Z 916.456,A -85,B 0,C 180,E1 22149.052,E2 22149.052} C_VEL
LIN {X 0,Y 195.539,Z 931.359,A -85,B 0,C 180,E1 22162.237,E2 22162.237} C_VEL
LIN {X 0,Y 195.467,Z 949.787,A -85,B 0,C 180,E1 22170.61,E2 22170.61} C_VEL
LIN {X 0,Y 167.652,Z 987.641,A -85,B 0,C 180,E1 22179.702,E2 22179.702} C_VEL
LIN {X 0,Y 142.523,Z 1013.911,A -85,B 0,C 180,E1 22196.014,E2 22196.014} C_VEL
LIN {X 0,Y 133.792,Z 1024.559,A -85,B 0,C 180,E1 22214.642,E2 22214.642} C_VEL
LIN {X 0,Y 134.575,Z 1025.768,A -85,B 0,C 180,E1 22226.769,E2 22226.769} C_VEL
LIN {X 0,Y 134.096,Z 1019.943,A -85,B 0,C 180,E1 22241.413,E2 22241.413} C_VEL
LIN {X 0,Y 140.72,Z 997.614,A -85,B 0,C 180,E1 22261.718,E2 22261.718} C_VEL
LIN {X 0,Y 157.706,Z 961.619,A -85,B 0,C 180,E1 22276.196,E2 22276.196} C_VEL
LIN {X 0,Y 169.259,Z 928.577,A -85,B 0,C 180,E1 22283.046,E2 22283.046} C_VEL
LIN {X 0,Y 161.078,Z 888.982,A -85,B 0,C 180,E1 22293.481,E2 22293.481} C_VEL
LIN {X 0,Y 145.749,Z 856.889,A -85,B 0,C 180,E1 22306.061,E2 22306.061} C_VEL
LIN {X 0,Y 134.911,Z 839.07,A -85,B 0,C 180,E1 22319.591,E2 22319.591} C_VEL
LIN {X 0,Y 130.53,Z 837.617,A -85,B 0,C 180,E1 22340.163,E2 22340.163} C_VEL
LIN {X 0,Y 133.895,Z 842.376,A -85,B 0,C 180,E1 22350.483,E2 22350.483} C_VEL
LIN {X 0,Y 143.711,Z 856.267,A -85,B 0,C 180,E1 22363.578,E2 22363.578} C_VEL
LIN {X 0,Y 156.688,Z 882.01,A -85,B 0,C 180,E1 22376.358,E2 22376.358} C_VEL
LIN {X 0,Y 162.865,Z 913.342,A -85,B 0,C 180,E1 22387.139,E2 22387.139} C_VEL
LIN {X 0,Y 159.53,Z 931.843,A -85,B 0,C 180,E1 22392.754,E2 22392.754} C_VEL
LIN {X 0,Y 144.529,Z 963.095,A -85,B 0,C 180,E1 22405.904,E2 22405.904} C_VEL
LIN {X 0,Y 136.262,Z 980.927,A -85,B 0,C 180,E1 22422.869,E2 22422.869} C_VEL
LIN {X 0,Y 136.844,Z 985.991,A -85,B 0,C 180,E1 22436.311,E2 22436.311} C_VEL
LIN {X 0,Y 136.913,Z 986.267,A -85,B 0,C 180,E1 22451.131,E2 22451.131} C_VEL
LIN {X 0,Y 157.826,Z 973.083,A -85,B 0,C 180,E1 22467.346,E2 22467.346} C_VEL
LIN {X 0,Y 179.945,Z 950.333,A -85,B 0,C 180,E1 22477.701,E2 22477.701} C_VEL
LIN {X 0,Y 185.672,Z 932.376,A -85,B 0,C 180,E1 22489.407,E2 22489.407} C_VEL
LIN {X 0,Y 187.95,Z 922.926,A -85,B 0,C 180,E1 22500.005,E2 22500.005} C_VEL
LIN {X 0,Y 188.977,Z 923.665,A -85,B 0,C 180,E1 22509.25,E2 22509.25} C_VEL
LIN {X 0,Y 190.619,Z 938.568,A -85,B 0,C 180,E1 22522.396,E2 22522.396} C_VEL
LIN {X 0,Y 189.55,Z 952.541,A -85,B 0,C 180,E1 22528.994,E2 22528.994} C_VEL
LIN {X 0,Y 161.322,Z 988.426,A -85,B 0,C 180,E1 22538.019,E2 22538.019} C_VEL
LIN {X 0,Y 135.806,Z 1012.954,A -85,B 0,C 180,E1 22554.082,E2 22554.082} C_VEL
LIN {X 0,Y 126.12,Z 1023.099,A -85,B 0,C 180,E1 22572.495,E2 22572.495} C_VEL
LIN {X 0,Y 126.589,Z 1024.479,A -85,B 0,C 180,E1 22586.565,E2 22586.565} C_VEL
LIN {X 0,Y 126.164,Z 1018.534,A -85,B 0,C 180,E1 22601.973,E2 22601.973} C_VEL
LIN {X 0,Y 133.169,Z 996.841,A -85,B 0,C 180,E1 22622.773,E2 22622.773} C_VEL
LIN {X 0,Y 151.024,Z 961.033,A -85,B 0,C 180,E1 22637.824,E2 22637.824} C_VEL
LIN {X 0,Y 162.492,Z 930.2,A -85,B 0,C 180,E1 22644.516,E2 22644.516} C_VEL
LIN {X 0,Y 155.338,Z 891.792,A -85,B 0,C 180,E1 22655.517,E2 22655.517} C_VEL
LIN {X 0,Y 141.198,Z 859.846,A -85,B 0,C 180,E1 22669.348,E2 22669.348} C_VEL
LIN {X 0,Y 132.571,Z 846.226,A -85,B 0,C 180,E1 22682.044,E2 22682.044} C_VEL
LIN {X 0,Y 130.375,Z 846.511,A -85,B 0,C 180,E1 22704.035,E2 22704.035} C_VEL
LIN {X 0,Y 139.836,Z 860.943,A -85,B 0,C 180,E1 22721.116,E2 22721.116} C_VEL
LIN {X 0,Y 152.071,Z 888.515,A -85,B 0,C 180,E1 22735.649,E2 22735.649} C_VEL
LIN {X 0,Y 156.38,Z 918.318,A -85,B 0,C 180,E1 22746.549,E2 22746.549} C_VEL
LIN {X 0,Y 151.043,Z 936.84,A -85,B 0,C 180,E1 22752.306,E2 22752.306} C_VEL
LIN {X 0,Y 135.482,Z 967.068,A -85,B 0,C 180,E1 22766.788,E2 22766.788} C_VEL
LIN {X 0,Y 127.857,Z 984.453,A -85,B 0,C 180,E1 22787.26,E2 22787.26} C_VEL
LIN {X 0,Y 134.703,Z 987.073,A -85,B 0,C 180,E1 22808.287,E2 22808.287} C_VEL
LIN {X 0,Y 136.913,Z 986.267,A -85,B 0,C 180,E1 22811.131,E2 22811.131} C_VEL
LIN {X 0,Y 144.662,Z 979.842,A -85,B 0,C 180,E1 22825.012,E2 22825.012} C_VEL
LIN {X 0,Y 172.248,Z 956.488,A -85,B 0,C 180,E1 22837.676,E2 22837.676} C_VEL
LIN {X 0,Y 179.601,Z 940.835,A -85,B 0,C 180,E1 22847.809,E2 22847.809} C_VEL
LIN {X 0,Y 183.458,Z 929.699,A -85,B 0,C 180,E1 22860.005,E2 22860.005} C_VEL
LIN {X 0,Y 184.551,Z 930.695,A -85,B 0,C 180,E1 22869.471,E2 22869.471} C_VEL
LIN {X 0,Y 185.31,Z 945.182,A -85,B 0,C 180,E1 22882.351,E2 22882.351} C_VEL
LIN {X 0,Y 184.077,Z 954.858,A -85,B 0,C 180,E1 22887.21,E2 22887.21} C_VEL
LIN {X 0,Y 153.844,Z 990.343,A -85,B 0,C 180,E1 22896.732,E2 22896.732} C_VEL
LIN {X 0,Y 127.679,Z 1013.32,A -85,B 0,C 180,E1 22913.54,E2 22913.54} C_VEL
LIN {X 0,Y 117.722,Z 1023.209,A -85,B 0,C 180,E1 22938.852,E2 22938.852} C_VEL
LIN {X 0,Y 118.816,Z 1021.481,A -85,B 0,C 180,E1 22953.663,E2 22953.663} C_VEL
LIN {X 0,Y 120.874,Z 1005.939,A -85,B 0,C 180,E1 22976.068,E2 22976.068} C_VEL
LIN {X 0,Y 135.978,Z 976.84,A -85,B 0,C 180,E1 22994.061,E2 22994.061} C_VEL
LIN {X 0,Y 155.282,Z 936.348,A -85,B 0,C 180,E1 23004.955,E2 23004.955} C_VEL
LIN {X 0,Y 151.814,Z 902.896,A -85,B 0,C 180,E1 23014.852,E2 23014.852} C_VEL
LIN {X 0,Y 140.694,Z 871.444,A -85,B 0,C 180,E1 23027.93,E2 23027.93} C_VEL
LIN {X 0,Y 131.387,Z 854.103,A -85,B 0,C 180,E1 23042.372,E2 23042.372} C_VEL
LIN {X 0,Y 129.363,Z 854.501,A -85,B 0,C 180,E1 23064.235,E2 23064.235} C_VEL
LIN {X 0,Y 137.588,Z 869.696,A -85,B 0,C 180,E1 23081.062,E2 23081.062} C_VEL
LIN {X 0,Y 147.307,Z 895.179,A -85,B 0,C 180,E1 23095.041,E2 23095.041} C_VEL
LIN {X 0,Y 149.594,Z 925.448,A -85,B 0,C 180,E1 23106.802,E2 23106.802} C_VEL
LIN {X 0,Y 132.764,Z 959.819,A -85,B 0,C 180,E1 23120.126,E2 23120.126} C_VEL
LIN {X 0,Y 121.196,Z 981.069,A -85,B 0,C 180,E1 23139.206,E2 23139.206} C_VEL
LIN {X 0,Y 120.867,Z 988.258,A -85,B 0,C 180,E1 23156.067,E2 23156.067} C_VEL
LIN {X 0,Y 134.364,Z 985.687,A -85,B 0,C 180,E1 23177.232,E2 23177.232} C_VEL
LIN {X 0,Y 144.662,Z 979.842,A -85,B 0,C 180,E1 23185.012,E2 23185.012} C_VEL
LIN {X 0,Y 158.049,Z 967.109,A -85,B 0,C 180,E1 23196.486,E2 23196.486} C_VEL
LIN {X 0,Y 168.633,Z 956.63,A -85,B 0,C 180,E1 23200.888,E2 23200.888} C_VEL
LIN {X 0,Y 175.968,Z 941.739,A -85,B 0,C 180,E1 23212.629,E2 23212.629} C_VEL
LIN {X 0,Y 179.356,Z 935.298,A -85,B 0,C 180,E1 23222.43,E2 23222.43} C_VEL
LIN {X 0,Y 179.84,Z 939.324,A -85,B 0,C 180,E1 23232.184,E2 23232.184} C_VEL
LIN {X 0,Y 179.31,Z 954.238,A -85,B 0,C 180,E1 23243.873,E2 23243.873} C_VEL
LIN {X 0,Y 175.342,Z 961.471,A -85,B 0,C 180,E1 23246.115,E2 23246.115} C_VEL
LIN {X 0,Y 144.451,Z 993.875,A -85,B 0,C 180,E1 23256.173,E2 23256.173} C_VEL
LIN {X 0,Y 118.074,Z 1014.682,A -85,B 0,C 180,E1 23274.666,E2 23274.666} C_VEL
LIN {X 0,Y 109.79,Z 1021.95,A -85,B 0,C 180,E1 23298.035,E2 23298.035} C_VEL
LIN {X 0,Y 110.838,Z 1020.087,A -85,B 0,C 180,E1 23313.927,E2 23313.927} C_VEL
LIN {X 0,Y 113.503,Z 1004.112,A -85,B 0,C 180,E1 23337.903,E2 23337.903} C_VEL
LIN {X 0,Y 130.395,Z 973.882,A -85,B 0,C 180,E1 23356.781,E2 23356.781} C_VEL
LIN {X 0,Y 149.163,Z 933.935,A -85,B 0,C 180,E1 23367.623,E2 23367.623} C_VEL
LIN {X 0,Y 144.618,Z 899.396,A -85,B 0,C 180,E1 23379.251,E2 23379.251} C_VEL
LIN {X 0,Y 134.635,Z 871.692,A -85,B 0,C 180,E1 23393.502,E2 23393.502} C_VEL
LIN {X 0,Y 129.1,Z 861.121,A -85,B 0,C 180,E1 23405.071,E2 23405.071} C_VEL
LIN {X 0,Y 128.5,Z 863.601,A -85,B 0,C 180,E1 23426.215,E2 23426.215} C_VEL
LIN {X 0,Y 136.069,Z 880.733,A -85,B 0,C 180,E1 23442.949,E2 23442.949} C_VEL
LIN {X 0,Y 142.899,Z 905.707,A -85,B 0,C 180,E1 23456.193,E2 23456.193} C_VEL
LIN {X 0,Y 142.122,Z 931.049,A -85,B 0,C 180,E1 23466.373,E2 23466.373} C_VEL
LIN {X 0,Y 124.036,Z 963.563,A -85,B 0,C 180,E1 23480.347,E2 23480.347} C_VEL
LIN {X 0,Y 112.622,Z 983.886,A -85,B 0,C 180,E1 23501.659,E2 23501.659} C_VEL
LIN {X 0,Y 116.751,Z 990.2,A -85,B 0,C 180,E1 23525.795,E2 23525.795} C_VEL
LIN {X 0,Y 137.103,Z 982.219,A -85,B 0,C 180,E1 23546.111,E2 23546.111} C_VEL
LIN {X 0,Y 158.049,Z 967.109,A -85,B 0,C 180,E1 23556.486,E2 23556.486} C_VEL
LIN {X 0,Y 164.398,Z 957.854,A -85,B 0,C 180,E1 23564.032,E2 23564.032} C_VEL
LIN {X 0,Y 171.932,Z 944.984,A -85,B 0,C 180,E1 23576.082,E2 23576.082} C_VEL
LIN {X 0,Y 174.378,Z 941.653,A -85,B 0,C 180,E1 23582.499,E2 23582.499} C_VEL
LIN {X 0,Y 174.693,Z 946.019,A -85,B 0,C 180,E1 23592.549,E2 23592.549} C_VEL
LIN {X 0,Y 173.329,Z 959.241,A -85,B 0,C 180,E1 23603.21,E2 23603.21} C_VEL
LIN {X 0,Y 139.573,Z 993.407,A -85,B 0,C 180,E1 23613.564,E2 23613.564} C_VEL
LIN {X 0,Y 111.463,Z 1013.699,A -85,B 0,C 180,E1 23632.219,E2 23632.219} C_VEL
LIN {X 0,Y 101.86,Z 1020.688,A -85,B 0,C 180,E1 23657.088,E2 23657.088} C_VEL
LIN {X 0,Y 102.842,Z 1018.68,A -85,B 0,C 180,E1 23674.233,E2 23674.233} C_VEL
LIN {X 0,Y 106.3,Z 1002.26,A -85,B 0,C 180,E1 23699.979,E2 23699.979} C_VEL
LIN {X 0,Y 124.126,Z 972.597,A -85,B 0,C 180,E1 23719.015,E2 23719.015} C_VEL
LIN {X 0,Y 142.639,Z 934.962,A -85,B 0,C 180,E1 23729.636,E2 23729.636} C_VEL
LIN {X 0,Y 138.683,Z 900.323,A -85,B 0,C 180,E1 23742.48,E2 23742.48} C_VEL
LIN {X 0,Y 130.369,Z 874.606,A -85,B 0,C 180,E1 23757.83,E2 23757.83} C_VEL
LIN {X 0,Y 126.547,Z 868.29,A -85,B 0,C 180,E1 23768.615,E2 23768.615} C_VEL
LIN {X 0,Y 126.739,Z 872.793,A -85,B 0,C 180,E1 23787.092,E2 23787.092} C_VEL
LIN {X 0,Y 133.029,Z 889.387,A -85,B 0,C 180,E1 23803.318,E2 23803.318} C_VEL
LIN {X 0,Y 137.511,Z 914.386,A -85,B 0,C 180,E1 23816.689,E2 23816.689} C_VEL
LIN {X 0,Y 134.664,Z 934.51,A -85,B 0,C 180,E1 23824.942,E2 23824.942} C_VEL
LIN {X 0,Y 115.48,Z 966.755,A -85,B 0,C 180,E1 23840.237,E2 23840.237} C_VEL
LIN {X 0,Y 104.502,Z 985.604,A -85,B 0,C 180,E1 23862.58,E2 23862.58} C_VEL
LIN {X 0,Y 110.033,Z 991.371,A -85,B 0,C 180,E1 23888.36,E2 23888.36} C_VEL
LIN {X 0,Y 132.571,Z 982.945,A -85,B 0,C 180,E1 23909.149,E2 23909.149} C_VEL
LIN {X 0,Y 162.754,Z 960.189,A -85,B 0,C 180,E1 23922.29,E2 23922.29} C_VEL
LIN {X 0,Y 164.398,Z 957.854,A -85,B 0,C 180,E1 23924.032,E2 23924.032} C_VEL
LIN {X 0,Y 166.222,Z 951.019,A -85,B 0,C 180,E1 23936.25,E2 23936.25} C_VEL
LIN {X 0,Y 169.112,Z 947.779,A -85,B 0,C 180,E1 23942.577,E2 23942.577} C_VEL
LIN {X 0,Y 169.209,Z 952.507,A -85,B 0,C 180,E1 23952.963,E2 23952.963} C_VEL
LIN {X 0,Y 166.474,Z 963.657,A -85,B 0,C 180,E1 23961.687,E2 23961.687} C_VEL
LIN {X 0,Y 131.967,Z 995.189,A -85,B 0,C 180,E1 23971.999,E2 23971.999} C_VEL
LIN {X 0,Y 101.856,Z 1014.596,A -85,B 0,C 180,E1 23993.427,E2 23993.427} C_VEL
LIN {X 0,Y 94.602,Z 1019.186,A -85,B 0,C 180,E1 24025.401,E2 24025.401} C_VEL
LIN {X 0,Y 94.518,Z 1013.326,A -85,B 0,C 180,E1 24043.937,E2 24043.937} C_VEL
LIN {X 0,Y 106.203,Z 989.815,A -85,B 0,C 180,E1 24071.368,E2 24071.368} C_VEL
LIN {X 0,Y 128.445,Z 953.921,A -85,B 0,C 180,E1 24087.296,E2 24087.296} C_VEL
LIN {X 0,Y 136.301,Z 935.29,A -85,B 0,C 180,E1 24092.095,E2 24092.095} C_VEL
LIN {X 0,Y 133.519,Z 903.441,A -85,B 0,C 180,E1 24105.041,E2 24105.041} C_VEL
LIN {X 0,Y 127.091,Z 880.299,A -85,B 0,C 180,E1 24120.581,E2 24120.581} C_VEL
LIN {X 0,Y 124.315,Z 875.878,A -85,B 0,C 180,E1 24130.544,E2 24130.544} C_VEL
LIN {X 0,Y 124.316,Z 880.302,A -85,B 0,C 180,E1 24146.389,E2 24146.389} C_VEL
LIN {X 0,Y 128.78,Z 895.221,A -85,B 0,C 180,E1 24161.783,E2 24161.783} C_VEL
LIN {X 0,Y 131.66,Z 918.134,A -85,B 0,C 180,E1 24174.999,E2 24174.999} C_VEL
LIN {X 0,Y 128.131,Z 936.575,A -85,B 0,C 180,E1 24182.971,E2 24182.971} C_VEL
LIN {X 0,Y 108.822,Z 967.112,A -85,B 0,C 180,E1 24197.924,E2 24197.924} C_VEL
LIN {X 0,Y 96.393,Z 987.309,A -85,B 0,C 180,E1 24223.658,E2 24223.658} C_VEL
LIN {X 0,Y 103.535,Z 992.537,A -85,B 0,C 180,E1 24251.266,E2 24251.266} C_VEL
LIN {X 0,Y 128.427,Z 983.649,A -85,B 0,C 180,E1 24272.4,E2 24272.4} C_VEL
LIN {X 0,Y 158.031,Z 962.397,A -85,B 0,C 180,E1 24284.83,E2 24284.83} C_VEL
LIN {X 0,Y 166.222,Z 951.019,A -85,B 0,C 180,E1 24296.25,E2 24296.25} C_VEL
LIN {X 0,Y 163.549,Z 954.099,A -85,B 0,C 180,E1 24304.474,E2 24304.474} C_VEL
LIN {X 0,Y 163.158,Z 960.403,A -85,B 0,C 180,E1 24315.209,E2 24315.209} C_VEL
LIN {X 0,Y 160.31,Z 966.962,A -85,B 0,C 180,E1 24319.741,E2 24319.741} C_VEL
LIN {X 0,Y 123.493,Z 997.428,A -85,B 0,C 180,E1 24330.664,E2 24330.664} C_VEL
LIN {X 0,Y 95.383,Z 1013.528,A -85,B 0,C 180,E1 24350.478,E2 24350.478} C_VEL
LIN {X 0,Y 86.611,Z 1017.831,A -85,B 0,C 180,E1 24384.976,E2 24384.976} C_VEL
LIN {X 0,Y 86.691,Z 1011.514,A -85,B 0,C 180,E1 24405.632,E2 24405.632} C_VEL
LIN {X 0,Y 100.033,Z 987.86,A -85,B 0,C 180,E1 24434.356,E2 24434.356} C_VEL
LIN {X 0,Y 123.74,Z 951.657,A -85,B 0,C 180,E1 24450.272,E2 24450.272} C_VEL
LIN {X 0,Y 130.099,Z 935.834,A -85,B 0,C 180,E1 24454.712,E2 24454.712} C_VEL
LIN {X 0,Y 128.298,Z 905.536,A -85,B 0,C 180,E1 24468.365,E2 24468.365} C_VEL
LIN {X 0,Y 123.788,Z 884.768,A -85,B 0,C 180,E1 24484.388,E2 24484.388} C_VEL
LIN {X 0,Y 121.526,Z 886.48,A -85,B 0,C 180,E1 24504.04,E2 24504.04} C_VEL
LIN {X 0,Y 124.672,Z 901.947,A -85,B 0,C 180,E1 24520.965,E2 24520.965} C_VEL
LIN {X 0,Y 125.621,Z 924.807,A -85,B 0,C 180,E1 24534.679,E2 24534.679} C_VEL
LIN {X 0,Y 121.62,Z 938.823,A -85,B 0,C 180,E1 24540.876,E2 24540.876} C_VEL
LIN {X 0,Y 99.973,Z 970.556,A -85,B 0,C 180,E1 24557.951,E2 24557.951} C_VEL
LIN {X 0,Y 88.342,Z 988.94,A -85,B 0,C 180,E1 24584.93,E2 24584.93} C_VEL
LIN {X 0,Y 98.629,Z 993.565,A -85,B 0,C 180,E1 24616.189,E2 24616.189} C_VEL
LIN {X 0,Y 127.294,Z 982.985,A -85,B 0,C 180,E1 24637.085,E2 24637.085} C_VEL
LIN {X 0,Y 153.141,Z 965.079,A -85,B 0,C 180,E1 24647.254,E2 24647.254} C_VEL
LIN {X 0,Y 161.951,Z 955.04,A -85,B 0,C 180,E1 24659.332,E2 24659.332} C_VEL
LIN {X 0,Y 163.549,Z 954.099,A -85,B 0,C 180,E1 24664.474,E2 24664.474} C_VEL
LIN {X 0,Y 158.33,Z 963.337,A -85,B 0,C 180,E1 24673.229,E2 24673.229} C_VEL
LIN {X 0,Y 156.616,Z 967.003,A -85,B 0,C 180,E1 24676.241,E2 24676.241} C_VEL
LIN {X 0,Y 130.175,Z 989.686,A -85,B 0,C 180,E1 24683.577,E2 24683.577} C_VEL
LIN {X 0,Y 93.236,Z 1010.667,A -85,B 0,C 180,E1 24702.912,E2 24702.912} C_VEL
LIN {X 0,Y 78.293,Z 1016.897,A -85,B 0,C 180,E1 24733.1,E2 24733.1} C_VEL
LIN {X 0,Y 78.87,Z 1014.282,A -85,B 0,C 180,E1 24755.523,E2 24755.523} C_VEL
LIN {X 0,Y 86.691,Z 995.409,A -85,B 0,C 180,E1 24789.39,E2 24789.39} C_VEL
LIN {X 0,Y 111.036,Z 962.436,A -85,B 0,C 180,E1 24809.628,E2 24809.628} C_VEL
LIN {X 0,Y 123.868,Z 939.07,A -85,B 0,C 180,E1 24816.416,E2 24816.416} C_VEL
LIN {X 0,Y 123.692,Z 910.528,A -85,B 0,C 180,E1 24830.28,E2 24830.28} C_VEL
LIN {X 0,Y 121.124,Z 893.636,A -85,B 0,C 180,E1 24843.585,E2 24843.585} C_VEL
LIN {X 0,Y 118.686,Z 891.996,A -85,B 0,C 180,E1 24858.636,E2 24858.636} C_VEL
LIN {X 0,Y 119.894,Z 904.437,A -85,B 0,C 180,E1 24876.624,E2 24876.624} C_VEL
LIN {X 0,Y 120.259,Z 925.018,A -85,B 0,C 180,E1 24890.891,E2 24890.891} C_VEL
LIN {X 0,Y 116.193,Z 939.607,A -85,B 0,C 180,E1 24898.087,E2 24898.087} C_VEL
LIN {X 0,Y 92.884,Z 971.681,A -85,B 0,C 180,E1 24915.812,E2 24915.812} C_VEL
LIN {X 0,Y 80.311,Z 990.561,A -85,B 0,C 180,E1 24946.463,E2 24946.463} C_VEL
LIN {X 0,Y 91.533,Z 994.867,A -85,B 0,C 180,E1 24978.248,E2 24978.248} C_VEL
LIN {X 0,Y 121.505,Z 985.015,A -85,B 0,C 180,E1 24999.503,E2 24999.503} C_VEL
LIN {X 0,Y 147.063,Z 969,A -85,B 0,C 180,E1 25008.604,E2 25008.604} C_VEL
LIN {X 0,Y 155.874,Z 960.666,A -85,B 0,C 180,E1 25019.397,E2 25019.397} C_VEL
LIN {X 0,Y 158.089,Z 960.762,A -85,B 0,C 180,E1 25028.285,E2 25028.285} C_VEL
LIN {X 0,Y 156.616,Z 967.003,A -85,B 0,C 180,E1 25036.241,E2 25036.241} C_VEL
LIN {X 0,Y 149.114,Z 973.802,A -85,B 0,C 180,E1 25037.478,E2 25037.478} C_VEL
LIN {X 0,Y 137.78,Z 981.495,A -85,B 0,C 180,E1 25037.541,E2 25037.541} C_VEL
LIN {X 0,Y 98.19,Z 1005.216,A -85,B 0,C 180,E1 25051.788,E2 25051.788} C_VEL
LIN {X 0,Y 73.593,Z 1014.852,A -85,B 0,C 180,E1 25078.97,E2 25078.97} C_VEL
LIN {X 0,Y 70.781,Z 1014.206,A -85,B 0,C 180,E1 25110.002,E2 25110.002} C_VEL
LIN {X 0,Y 74.536,Z 1001.103,A -85,B 0,C 180,E1 25143.028,E2 25143.028} C_VEL
LIN {X 0,Y 97.872,Z 972.041,A -85,B 0,C 180,E1 25168.52,E2 25168.52} C_VEL
LIN {X 0,Y 117.752,Z 941.662,A -85,B 0,C 180,E1 25178.547,E2 25178.547} C_VEL
LIN {X 0,Y 118.988,Z 915.022,A -85,B 0,C 180,E1 25192.564,E2 25192.564} C_VEL
LIN {X 0,Y 117.552,Z 899.352,A -85,B 0,C 180,E1 25206.744,E2 25206.744} C_VEL
LIN {X 0,Y 115.406,Z 901.452,A -85,B 0,C 180,E1 25223.227,E2 25223.227} C_VEL
LIN {X 0,Y 115.769,Z 915.172,A -85,B 0,C 180,E1 25239.329,E2 25239.329} C_VEL
LIN {X 0,Y 112.823,Z 936.928,A -85,B 0,C 180,E1 25253.573,E2 25253.573} C_VEL
LIN {X 0,Y 88.389,Z 970.041,A -85,B 0,C 180,E1 25270.764,E2 25270.764} C_VEL
LIN {X 0,Y 72.74,Z 990.191,A -85,B 0,C 180,E1 25302.04,E2 25302.04} C_VEL
LIN {X 0,Y 78.789,Z 996.249,A -85,B 0,C 180,E1 25332.384,E2 25332.384} C_VEL
LIN {X 0,Y 106.616,Z 990.819,A -85,B 0,C 180,E1 25357.693,E2 25357.693} C_VEL
LIN {X 0,Y 141.883,Z 972.107,A -85,B 0,C 180,E1 25370.773,E2 25370.773} C_VEL
LIN {X 0,Y 149.905,Z 965.774,A -85,B 0,C 180,E1 25380.006,E2 25380.006} C_VEL
LIN {X 0,Y 151.935,Z 966.309,A -85,B 0,C 180,E1 25388.623,E2 25388.623} C_VEL
LIN {X 0,Y 149.392,Z 971.998,A -85,B 0,C 180,E1 25395.204,E2 25395.204} C_VEL
LIN {X 0,Y 137.78,Z 981.495,A -85,B 0,C 180,E1 25397.541,E2 25397.541} C_VEL
LIN {X 0,Y 107.68,Z 998.033,A -85,B 0,C 180,E1 25401.702,E2 25401.702} C_VEL
LIN {X 0,Y 73.573,Z 1011.74,A -85,B 0,C 180,E1 25423.79,E2 25423.79} C_VEL
LIN {X 0,Y 62.593,Z 1013.74,A -85,B 0,C 180,E1 25463.04,E2 25463.04} C_VEL
LIN {X 0,Y 62.854,Z 1008.737,A -85,B 0,C 180,E1 25485.7,E2 25485.7} C_VEL
LIN {X 0,Y 79.335,Z 986.405,A -85,B 0,C 180,E1 25522.099,E2 25522.099} C_VEL
LIN {X 0,Y 107.564,Z 951.145,A -85,B 0,C 180,E1 25539.047,E2 25539.047} C_VEL
LIN {X 0,Y 112.574,Z 939.633,A -85,B 0,C 180,E1 25543.242,E2 25543.242} C_VEL
LIN {X 0,Y 114.389,Z 915.128,A -85,B 0,C 180,E1 25558.316,E2 25558.316} C_VEL
LIN {X 0,Y 114.333,Z 907.697,A -85,B 0,C 180,E1 25565.438,E2 25565.438} C_VEL
LIN {X 0,Y 112.163,Z 907.361,A -85,B 0,C 180,E1 25579.763,E2 25579.763} C_VEL
LIN {X 0,Y 111.107,Z 919.562,A -85,B 0,C 180,E1 25596.609,E2 25596.609} C_VEL
LIN {X 0,Y 107.352,Z 938.81,A -85,B 0,C 180,E1 25610.495,E2 25610.495} C_VEL
LIN {X 0,Y 81.459,Z 971.564,A -85,B 0,C 180,E1 25628.123,E2 25628.123} C_VEL
LIN {X 0,Y 64.634,Z 991.874,A -85,B 0,C 180,E1 25663.577,E2 25663.577} C_VEL
LIN {X 0,Y 72.803,Z 997.497,A -85,B 0,C 180,E1 25696.846,E2 25696.846} C_VEL
LIN {X 0,Y 103.695,Z 991.647,A -85,B 0,C 180,E1 25722.032,E2 25722.032} C_VEL
LIN {X 0,Y 137.162,Z 974.952,A -85,B 0,C 180,E1 25733.423,E2 25733.423} C_VEL
LIN {X 0,Y 145.184,Z 969.931,A -85,B 0,C 180,E1 25743.002,E2 25743.002} C_VEL
LIN {X 0,Y 144.816,Z 973.463,A -85,B 0,C 180,E1 25751.894,E2 25751.894} C_VEL
LIN {X 0,Y 107.68,Z 998.033,A -85,B 0,C 180,E1 25761.702,E2 25761.702} C_VEL
LIN {X 0,Y 76.927,Z 1008.15,A -85,B 0,C 180,E1 25770.844,E2 25770.844} C_VEL
LIN {X 0,Y 54.378,Z 1012.602,A -85,B 0,C 180,E1 25817.712,E2 25817.712} C_VEL
LIN {X 0,Y 54.918,Z 1009.818,A -85,B 0,C 180,E1 25837.945,E2 25837.945} C_VEL
LIN {X 0,Y 69.467,Z 989.246,A -85,B 0,C 180,E1 25882.366,E2 25882.366} C_VEL
LIN {X 0,Y 99.163,Z 955.904,A -85,B 0,C 180,E1 25901.249,E2 25901.249} C_VEL
LIN {X 0,Y 106.749,Z 943.024,A -85,B 0,C 180,E1 25905.496,E2 25905.496} C_VEL
LIN {X 0,Y 110.041,Z 920.443,A -85,B 0,C 180,E1 25920.458,E2 25920.458} C_VEL
LIN {X 0,Y 110.158,Z 914.204,A -85,B 0,C 180,E1 25927.911,E2 25927.911} C_VEL
LIN {X 0,Y 107.819,Z 916.634,A -85,B 0,C 180,E1 25943.809,E2 25943.809} C_VEL
LIN {X 0,Y 105.333,Z 930.422,A -85,B 0,C 180,E1 25959.655,E2 25959.655} C_VEL
LIN {X 0,Y 100.28,Z 944.062,A -85,B 0,C 180,E1 25968.698,E2 25968.698} C_VEL
LIN {X 0,Y 73.031,Z 974.659,A -85,B 0,C 180,E1 25986.629,E2 25986.629} C_VEL
LIN {X 0,Y 56.66,Z 993.078,A -85,B 0,C 180,E1 26023.808,E2 26023.808} C_VEL
LIN {X 0,Y 73.009,Z 998.595,A -85,B 0,C 180,E1 26068.703,E2 26068.703} C_VEL
LIN {X 0,Y 111.771,Z 988.522,A -85,B 0,C 180,E1 26090.367,E2 26090.367} C_VEL
LIN {X 0,Y 133.161,Z 977.54,A -85,B 0,C 180,E1 26096.74,E2 26096.74} C_VEL
LIN {X 0,Y 138.562,Z 974.781,A -85,B 0,C 180,E1 26103.146,E2 26103.146} C_VEL
LIN {X 0,Y 137.318,Z 977.983,A -85,B 0,C 180,E1 26110.33,E2 26110.33} C_VEL
LIN {X 0,Y 93.832,Z 1002.161,A -85,B 0,C 180,E1 26121.578,E2 26121.578} C_VEL
LIN {X 0,Y 76.927,Z 1008.15,A -85,B 0,C 180,E1 26130.844,E2 26130.844} C_VEL
LIN {X 0,Y 50.75,Z 1011.417,A -85,B 0,C 180,E1 26152.618,E2 26152.618} C_VEL
LIN {X 0,Y 47.083,Z 1009.917,A -85,B 0,C 180,E1 26190.003,E2 26190.003} C_VEL
LIN {X 0,Y 56.458,Z 994.643,A -85,B 0,C 180,E1 26238.399,E2 26238.399} C_VEL
LIN {X 0,Y 87.548,Z 964.151,A -85,B 0,C 180,E1 26262.438,E2 26262.438} C_VEL
LIN {X 0,Y 101.382,Z 944.961,A -85,B 0,C 180,E1 26268.796,E2 26268.796} C_VEL
LIN {X 0,Y 105.867,Z 924.201,A -85,B 0,C 180,E1 26284.102,E2 26284.102} C_VEL
LIN {X 0,Y 105.53,Z 920.511,A -85,B 0,C 180,E1 26292.449,E2 26292.449} C_VEL
LIN {X 0,Y 102.769,Z 926.348,A -85,B 0,C 180,E1 26308.042,E2 26308.042} C_VEL
LIN {X 0,Y 97.836,Z 941.49,A -85,B 0,C 180,E1 26322.513,E2 26322.513} C_VEL
LIN {X 0,Y 80.408,Z 962.793,A -85,B 0,C 180,E1 26332.164,E2 26332.164} C_VEL
LIN {X 0,Y 53.589,Z 987.722,A -85,B 0,C 180,E1 26362.271,E2 26362.271} C_VEL
LIN {X 0,Y 54.691,Z 999.31,A -85,B 0,C 180,E1 26416.096,E2 26416.096} C_VEL
LIN {X 0,Y 86.129,Z 997.131,A -85,B 0,C 180,E1 26445.704,E2 26445.704} C_VEL
LIN {X 0,Y 125.71,Z 982.083,A -85,B 0,C 180,E1 26458.198,E2 26458.198} C_VEL
LIN {X 0,Y 131.682,Z 979.346,A -85,B 0,C 180,E1 26463.31,E2 26463.31} C_VEL
LIN {X 0,Y 128.355,Z 982.679,A -85,B 0,C 180,E1 26468.047,E2 26468.047} C_VEL
LIN {X 0,Y 82.911,Z 1004.198,A -85,B 0,C 180,E1 26480.056,E2 26480.056} C_VEL
LIN {X 0,Y 50.75,Z 1011.417,A -85,B 0,C 180,E1 26512.618,E2 26512.618} C_VEL
LIN {X 0,Y 40.086,Z 1009.312,A -85,B 0,C 180,E1 26544.067,E2 26544.067} C_VEL
LIN {X 0,Y 38.857,Z 1007.359,A -85,B 0,C 180,E1 26556.921,E2 26556.921} C_VEL
LIN {X 0,Y 56.443,Z 988.569,A -85,B 0,C 180,E1 26610.91,E2 26610.91} C_VEL
LIN {X 0,Y 89.8,Z 956.338,A -85,B 0,C 180,E1 26629.176,E2 26629.176} C_VEL
LIN {X 0,Y 96.5,Z 946.294,A -85,B 0,C 180,E1 26632.833,E2 26632.833} C_VEL
LIN {X 0,Y 101.545,Z 929.333,A -85,B 0,C 180,E1 26646.643,E2 26646.643} C_VEL
LIN {X 0,Y 100.226,Z 928.194,A -85,B 0,C 180,E1 26657.624,E2 26657.624} C_VEL
LIN {X 0,Y 95.781,Z 938.358,A -85,B 0,C 180,E1 26673.67,E2 26673.67} C_VEL
LIN {X 0,Y 89.711,Z 949.053,A -85,B 0,C 180,E1 26681.351,E2 26681.351} C_VEL
LIN {X 0,Y 57.958,Z 979.379,A -85,B 0,C 180,E1 26700.595,E2 26700.595} C_VEL
LIN {X 0,Y 40.711,Z 996.633,A -85,B 0,C 180,E1 26751.317,E2 26751.317} C_VEL
LIN {X 0,Y 62.245,Z 1001.105,A -85,B 0,C 180,E1 26798.563,E2 26798.563} C_VEL
LIN {X 0,Y 102.558,Z 992.869,A -85,B 0,C 180,E1 26817.149,E2 26817.149} C_VEL
LIN {X 0,Y 120.555,Z 985.265,A -85,B 0,C 180,E1 26821.114,E2 26821.114} C_VEL
LIN {X 0,Y 124.808,Z 983.627,A -85,B 0,C 180,E1 26824.198,E2 26824.198} C_VEL
LIN {X 0,Y 78.653,Z 1003.784,A -85,B 0,C 180,E1 26835.275,E2 26835.275} C_VEL
LIN {X 0,Y 41.139,Z 1010.338,A -85,B 0,C 180,E1 26876.409,E2 26876.409} C_VEL
LIN {X 0,Y 38.857,Z 1007.359,A -85,B 0,C 180,E1 26916.921,E2 26916.921} C_VEL
LIN {X 0,Y 41.293,Z 994.795,A -85,B 0,C 180,E1 26965.942,E2 26965.942} C_VEL
LIN {X 0,Y 76.816,Z 966.084,A -85,B 0,C 180,E1 26991.046,E2 26991.046} C_VEL
LIN {X 0,Y 91.472,Z 949.049,A -85,B 0,C 180,E1 26996.276,E2 26996.276} C_VEL
LIN {X 0,Y 97.075,Z 934.522,A -85,B 0,C 180,E1 27009.439,E2 27009.439} C_VEL
LIN {X 0,Y 93.784,Z 937.619,A -85,B 0,C 180,E1 27023.853,E2 27023.853} C_VEL
LIN {X 0,Y 87.266,Z 949.04,A -85,B 0,C 180,E1 27036.425,E2 27036.425} C_VEL
LIN {X 0,Y 52.448,Z 980.422,A -85,B 0,C 180,E1 27054.638,E2 27054.638} C_VEL
LIN {X 0,Y 33.083,Z 998.224,A -85,B 0,C 180,E1 27116.574,E2 27116.574} C_VEL
LIN {X 0,Y 55.511,Z 1002.451,A -85,B 0,C 180,E1 27163.092,E2 27163.092} C_VEL
LIN {X 0,Y 98.653,Z 994.933,A -85,B 0,C 180,E1 27181.031,E2 27181.031} C_VEL
LIN {X 0,Y 105.639,Z 992.509,A -85,B 0,C 180,E1 27182.499,E2 27182.499} C_VEL
LIN {X 0,Y 56.107,Z 1007.261,A -85,B 0,C 180,E1 27198.808,E2 27198.808} C_VEL
LIN {X 0,Y 30.846,Z 1008.017,A -85,B 0,C 180,E1 27255.765,E2 27255.765} C_VEL
LIN {X 0,Y 32.068,Z 1002.713,A -85,B 0,C 180,E1 27298.25,E2 27298.25} C_VEL
LIN {X 0,Y 41.293,Z 994.795,A -85,B 0,C 180,E1 27325.942,E2 27325.942} C_VEL
LIN {X 0,Y 61.139,Z 976.434,A -85,B 0,C 180,E1 27352.562,E2 27352.562} C_VEL
LIN {X 0,Y 86.934,Z 951.241,A -85,B 0,C 180,E1 27360.441,E2 27360.441} C_VEL
LIN {X 0,Y 91.79,Z 941.445,A -85,B 0,C 180,E1 27369.507,E2 27369.507} C_VEL
LIN {X 0,Y 88.529,Z 943.991,A -85,B 0,C 180,E1 27383.12,E2 27383.12} C_VEL
LIN {X 0,Y 82.442,Z 952.324,A -85,B 0,C 180,E1 27391.892,E2 27391.892} C_VEL
LIN {X 0,Y 46.027,Z 982.505,A -85,B 0,C 180,E1 27408.741,E2 27408.741} C_VEL
LIN {X 0,Y 26.249,Z 1000.056,A -85,B 0,C 180,E1 27487.431,E2 27487.431} C_VEL
LIN {X 0,Y 54.027,Z 1003.62,A -85,B 0,C 180,E1 27531.942,E2 27531.942} C_VEL
LIN {X 0,Y 81.103,Z 1000.509,A -85,B 0,C 180,E1 27542.194,E2 27542.194} C_VEL
LIN {X 0,Y 40.395,Z 1007.473,A -85,B 0,C 180,E1 27560.097,E2 27560.097} C_VEL
LIN {X 0,Y 22.989,Z 1004.721,A -85,B 0,C 180,E1 27637.744,E2 27637.744} C_VEL
LIN {X 0,Y 50.558,Z 984.363,A -85,B 0,C 180,E1 27707.309,E2 27707.309} C_VEL
LIN {X 0,Y 61.139,Z 976.434,A -85,B 0,C 180,E1 27712.562,E2 27712.562} C_VEL
LIN {X 0,Y 75.057,Z 961.53,A -85,B 0,C 180,E1 27723.276,E2 27723.276} C_VEL
LIN {X 0,Y 82.914,Z 953.181,A -85,B 0,C 180,E1 27725.24,E2 27725.24} C_VEL
LIN {X 0,Y 86.155,Z 947.886,A -85,B 0,C 180,E1 27730.373,E2 27730.373} C_VEL
LIN {X 0,Y 82.849,Z 950.313,A -85,B 0,C 180,E1 27742.377,E2 27742.377} C_VEL
LIN {X 0,Y 78.442,Z 955.242,A -85,B 0,C 180,E1 27746.831,E2 27746.831} C_VEL
LIN {X 0,Y 40.275,Z 984.581,A -85,B 0,C 180,E1 27761.092,E2 27761.092} C_VEL
LIN {X 0,Y 19.811,Z 1001.418,A -85,B 0,C 180,E1 27859.986,E2 27859.986} C_VEL
LIN {X 0,Y 53.138,Z 1004.957,A -85,B 0,C 180,E1 27901.833,E2 27901.833} C_VEL
LIN {X 0,Y 15.012,Z 1004.304,A -85,B 0,C 180,E1 27981.692,E2 27981.692} C_VEL
LIN {X 0,Y 42.004,Z 986.843,A -85,B 0,C 180,E1 28073.51,E2 28073.51} C_VEL
LIN {X 0,Y 75.057,Z 961.53,A -85,B 0,C 180,E1 28083.276,E2 28083.276} C_VEL
LIN {X 0,Y 79.27,Z 955.206,A -85,B 0,C 180,E1 28090.724,E2 28090.724} C_VEL
LIN {X 0,Y 78.26,Z 955.089,A -85,B 0,C 180,E1 28098.789,E2 28098.789} C_VEL
LIN {X 0,Y 69.592,Z 963.141,A -85,B 0,C 180,E1 28102.058,E2 28102.058} C_VEL
LIN {X 0,Y 27.981,Z 990.391,A -85,B 0,C 180,E1 28115.549,E2 28115.549} C_VEL
LIN {X 0,Y 22.831,Z 1004.27,A -85,B 0,C 180,E1 28255.476,E2 28255.476} C_VEL
LIN {X 0,Y 27.806,Z 1004.974,A -85,B 0,C 180,E1 28259.869,E2 28259.869} C_VEL
LIN {X 0,Y 7.548,Z 1001.362,A -85,B 0,C 180,E1 28380.197,E2 28380.197} C_VEL
LIN {X 0,Y 49.625,Z 979.898,A -85,B 0,C 180,E1 28446.33,E2 28446.33} C_VEL
LIN {X 0,Y 79.387,Z 955.085,A -85,B 0,C 180,E1 28450.618,E2 28450.618} C_VEL
LIN {X 0,Y 78.26,Z 955.089,A -85,B 0,C 180,E1 28458.789,E2 28458.789} C_VEL
LIN {X 0,Y 68.741,Z 963.902,A -85,B 0,C 180,E1 28462.625,E2 28462.625} C_VEL
LIN {X 0,Y 45.392,Z 981.225,A -85,B 0,C 180,E1 28457.059,E2 28457.059} C_VEL
LIN {X 0,Y 8.009,Z 998.516,A -85,B 0,C 180,E1 28458.605,E2 28458.605} C_VEL
LIN {X 0,Y 52.631,Z 976.668,A -85,B 0,C 180,E1 28455.564,E2 28455.564} C_VEL
LIN {X 0,Y 55.406,Z 974.636,A -85,B 0,C 180,E1 28456.528,E2 28456.528} C_VEL
LIN {X 0,Y 45.392,Z 981.225,A -85,B 0,C 180,E1 28457.059,E2 28457.059} C_VEL
LIN {X 0,Y 44.418,Z 982.943,A -85,B 0,C 180,E1 28457.117,E2 28457.117} C_VEL
LIN {X 0,Y 44.418,Z 1084,A -85,B 0,C 180,E1 28457.117,E2 28457.117} C_VEL
LIN {X 0,Y 44.418,Z 1084,A -85,B 0,C 180,E1 28457.117,E2 28457.117}

